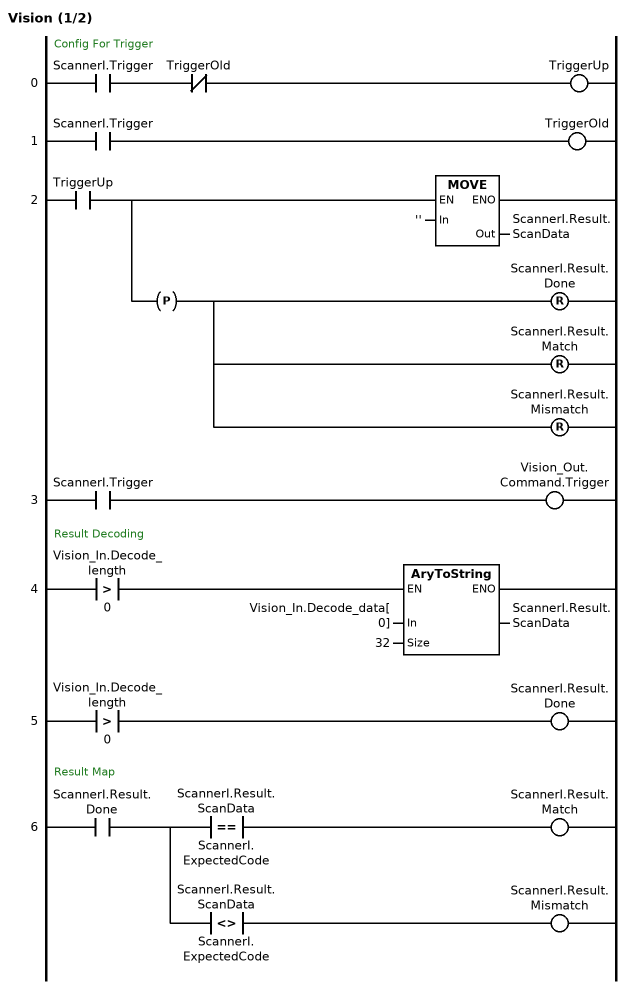
(* Rung 0: Config For Trigger *)
TriggerUp := ScannerI.Trigger AND NOT TriggerOld;
(* Rung 1 *)
TriggerOld := ScannerI.Trigger;
(* Rung 2 *)
IF TriggerUp THEN ScannerI.Result.ScanData := ''; END_IF;
_e1(CLK := TriggerUp);
IF _e1.Q THEN
    ScannerI.Result.Done := FALSE;
    ScannerI.Result.Match := FALSE;
    ScannerI.Result.Mismatch := FALSE;
END_IF;
(* Rung 3 *)
Vision_Out.Command.Trigger := ScannerI.Trigger;
(* Rung 4: Result Decoding *)
IF Vision_In.Decode_length > 0 THEN
    ScannerI.Result.ScanData := AryToString(In := Vision_In.Decode_data[0], Size := 32);
END_IF;
(* Rung 5 *)
ScannerI.Result.Done := Vision_In.Decode_length > 0;
(* Rung 6: Result Map *)
_p2 := ScannerI.Result.Done;
ScannerI.Result.Match := ScannerI.Result.Done AND (ScannerI.Result.ScanData = ScannerI.ExpectedCode);
ScannerI.Result.Mismatch := _p2 AND (ScannerI.Result.ScanData <> ScannerI.ExpectedCode);

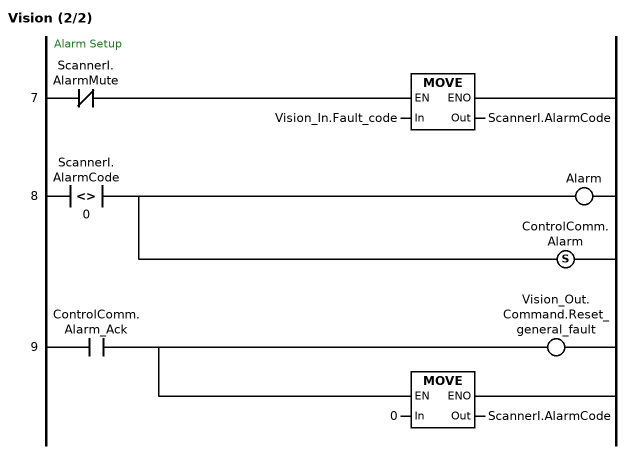
(* Rung 7: Alarm Setup *)
IF NOT ScannerI.AlarmMute THEN ScannerI.AlarmCode := Vision_In.Fault_code; END_IF;
(* Rung 8 *)
Alarm := ScannerI.AlarmCode <> 0;
IF ScannerI.AlarmCode <> 0 THEN ControlComm.Alarm := TRUE; END_IF;
(* Rung 9 *)
Vision_Out.Command.Reset_general_fault := ControlComm.Alarm_Ack;
IF ControlComm.Alarm_Ack THEN ScannerI.AlarmCode := 0; END_IF;
END_FUNCTION_BLOCK